(*			
	RafalOS
	Rafał Osajda		12.11.2025		TC 4024.66
	interfejs potrzebny w HMI
*)
INTERFACE ITF_HMIEButton_HMI EXTENDS ITF_BaseComponent_HMI

END_INTERFACE

(* stored: Version 1.1.0.1
   Itf ITF_HMIEButton_HMI: Id {02f9390e-52b4-0016-1a97-38f0c6617069} *)
